{attribute 'qualified_only'}
VAR_GLOBAL CONSTANT
  //do_LibTest : BOOL := TRUE;
  //do_TestStartUp : BOOL := TRUE;
END_VAR

(* stored: Version 1.1.0.1, ProductVersion 3.1.4024.3
   GVL GVL_TestCfg: Id {cd9ee570-7c80-458a-bd9b-3c5c2bf2c812}, ParameterList True *)
